FUNCTION_BLOCK BigComputation
  (* Version 1.0, 2005-12-19, Goran Cengic, Chalmers *)
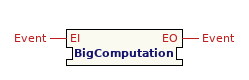
  EVENT_INPUT
    EI;
  END_EVENT
  EVENT_OUTPUT
    EO;
  END_EVENT
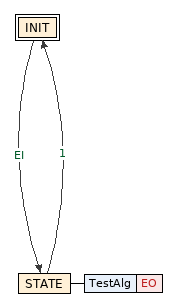
  EC_STATES
    INIT;
    STATE : TestAlg -> EO;
  END_STATES
  EC_TRANSITIONS
    INIT TO STATE := EI;
    STATE TO INIT := 1;
  END_TRANSITIONS
  ALGORITHM TestAlg IN Java:
	for (int i = 0; i < 1000000;)
	{
	   i = i + 1;
	}
	System.out.println("TestAlg: done.");
  END_ALGORITHM
END_FUNCTION_BLOCK
